FUNCTION_BLOCK FB_ReactorTemperatureControlStateMachine
VAR_INPUT
	temperatureMeasurement : REAL;
	temperatureSetpoint : REAL;
	pidParameters : ST_PidParameters;
	manualControlPercentage : INT;
	autoControlSelected : BOOL;
END_VAR
VAR_OUTPUT
	relayOn : BOOL;
END_VAR
VAR
	ReactorTemperaturePIDControl : FB_PidControllerRelayOutput;
END_VAR


// Monitor PID controller parameters
ReactorTemperaturePIDControl.SetParameters(parameters := pidParameters);

// Control logic according to mode selection
IF autoControlSelected THEN
	ReactorTemperaturePIDControl.AutomaticControl(processVariable := temperatureMeasurement,
												setpoint := temperatureSetpoint);													
ELSIF NOT autoControlSelected AND manualControlPercentage > 0 THEN
	ReactorTemperaturePIDControl.ManualControl(iControlPercentage := manualControlPercentage);
ELSE
	ReactorTemperaturePIDControl.ResetControl();
END_IF

// Control temperature relay 
relayOn := ReactorTemperaturePIDControl.relayOn;

END_FUNCTION_BLOCK

(* stored: Version 1.1.0.1, ProductVersion 3.1.4024.9
   POU FB_ReactorTemperatureControlStateMachine: Id {a4816a41-d106-4c43-933b-fcb27a662bd9}, SpecialFunc None *)
